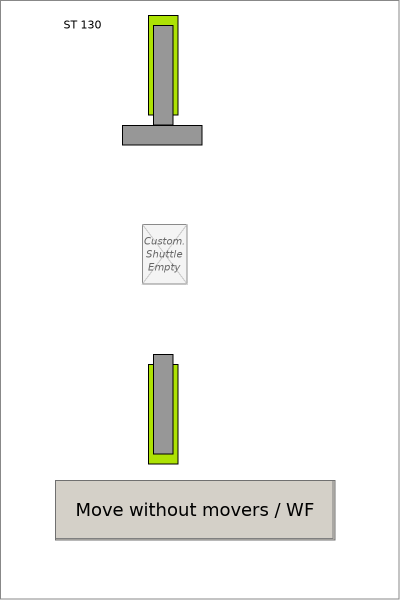
VISUALIZATION VISU_ST130  // 400x600
    Image (142,224 45x60), invisible if: NOT __ISVALIDREF(GVL.st130_aut._Mover), image: Custom.Shuttle Empty
    Rectangle (148,15 30x100)
    Rectangle (153,25 20x100)
        p2738717112: GVL.st130_aut.fb_Dose.fb_simu_axis130_01Z.rOUT_PixActual
    Label (40,15 85x20), "ST 130"
    Rectangle (122,125 80x20)
        p2738717112: GVL.st130_aut.fb_Dose.fb_simu_axis130_01Z.rOUT_PixActual
    Rectangle (148,364 30x100)
    Rectangle (153,354 20x100)
        p2738717112: -GVL.st130_aut.fb_Dose.fb_simu_axis130_10Z.rOUT_PixActual
    Button (55,480 280x60), "Move without movers / WF", colour toggle: HMI.bArForceCyclusState[StationList_e.ST130]
        tap HMI.btArForceCyclus[StationList_e.ST130].button
END_VISUALIZATION

(* stored: Version 1.1.0.1, ProductVersion 3.1.4024.6
   Visu VISU_ST130: Id {1f177acf-ab7c-4e65-84d9-7e74544c4919} *)
